// Mitsubishi GX Works2 project: LAB3 CODE   PLC: FX1S
// LAB3

PROGRAM MAIN
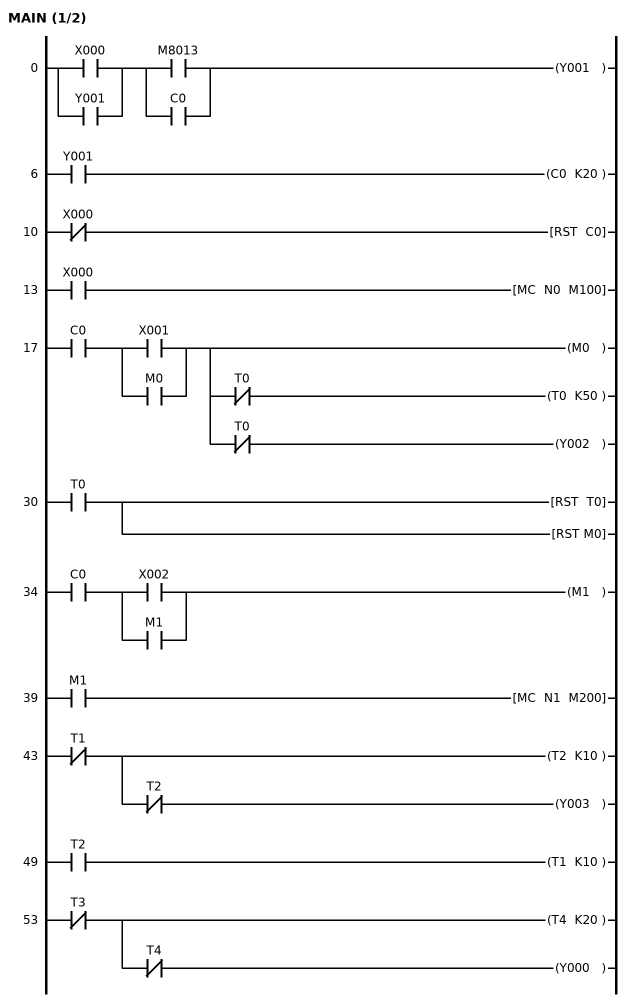
0     LD      X000
      OR      Y001
      LD      M8013
      OR      C0
      ANB
      OUT     Y001
6     LD      Y001
      OUT     C0 K20
10    LDI     X000
      RST     C0
13    LD      X000
      MC      N0 M100
17    LD      C0
      LD      X001
      OR      M0
      ANB
      OUT     M0
      MPS
      ANI     T0
      OUT     T0 K50
      MPP
      ANI     T0
      OUT     Y002
30    LD      T0
      RST     T0
      RST     M0
34    LD      C0
      LD      X002
      OR      M1
      ANB
      OUT     M1
39    LD      M1
      MC      N1 M200
43    LDI     T1
      OUT     T2 K10
      ANI     T2
      OUT     Y003
49    LD      T2
      OUT     T1 K10
53    LDI     T3
      OUT     T4 K20
      ANI     T4
      OUT     Y000
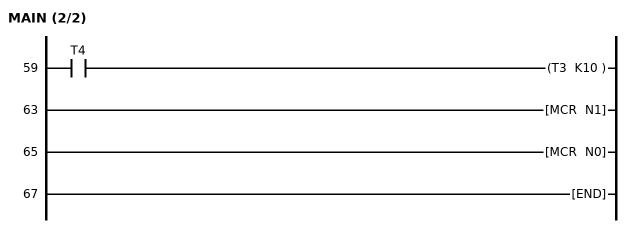
59    LD      T4
      OUT     T3 K10
63    MCR     N1
65    MCR     N0
67    END
END_PROGRAM
